// TIA Portal V17 export
// export: Created 2026-07-06T15:33:04.7365768Z, ExportSetting WithDefaults, DisplayName Totally Integrated Automation Portal, DisplayVersion V17, DisplayName TIA Portal Openness, DisplayVersion V17, DisplayName TIA Portal Version Control Interface, DisplayVersion V17, DisplayName STEP 7 Professional, DisplayVersion V17, DisplayName STEP 7 Safety, DisplayVersion V17, DisplayName WinCC Professional, DisplayVersion V17
DATA_BLOCK "Right_motor_DB"   // DB10
VERSION : 0.1
// stored: AutoNumber true, DBAccessibleFromOPCUA true, InstanceOfName Kinco_CAN_Data, InstanceOfType FB
"Kinco_CAN_Data"
   // VAR_INPUT
   //    Wake_node_trig : Bool;
   //    Op_mode_in : Byte;
   //    Control_word : Word;
   //    Target_RPM : DInt;
   //    Target_pos : DInt;
   //    profile_speed : DInt;
   //    Node_ID : Int;
   //    connection_established : Bool;
   //    send_pulse : Bool;
   //    move_pulse : Bool;
   //    Data_Recv { ExternalAccessible := 'False'; ExternalVisible := 'False'; ExternalWritable := 'False'} : Array[0..12] of Byte;
   // END_VAR
   // VAR_OUTPUT
   //    speed_real : DInt;
   //    pos_act : DInt;
   //    current : Real;
   //    status_word : Word;
   //    error_state : Word;
   //    Op_mode : Byte;
   //    Intial_state : Bool;
   //    Pre_operational_state : Bool;
   //    Operation_state : Bool;
   //    Stop_state : Bool;
   // END_VAR
   // VAR_IN_OUT
   //    Data_to_be_sent : Array[0..12] of Byte;
   // END_VAR
   // VAR
   //    tsend_inst : TSEND;
   //    Target_RPM_hex { S7_SetPoint := 'True'} : DWord;
   //    Target_pos_hex : DWord;
   //    profile_speed_hex : DWord;
   // END_VAR
BEGIN
END_DATA_BLOCK
